// TwinCAT 3 PLC project Untitled1
// ProgramVersion: 3.1.4024.0
// libraries:
//   Tc2_Standard, * (Beckhoff Automation GmbH)
//   Tc2_System, * (Beckhoff Automation GmbH)
//   Tc3_Module, * (Beckhoff Automation GmbH)
//   VisuSymbols,3.5.10.0,System
// project tree:
//   DUTs/ T_State.TcDUT
//   / GlobalTextList.TcGTLO (not stored), PlcTask.TcTTO (not stored), task1.TcTTO (not stored), task2.TcTTO (not stored), task3.TcTTO (not stored), Task_4.TcTTO, Visualization Manager.TcVMO (not stored), Visualization.TcVIS (not stored)
//   GVLs/ GVL.TcGVL
//   POUs/ Main.TcPOU (not stored), PRG_BeerSession.TcPOU, PRG_GameSession.TcPOU, PRG_TrainTrip.TcPOU
// real-time tasks:
//   TASK PlcTask: cycle T#10ms, priority 20, ADS port 350
//   TASK Task 4: cycle T#10ms, priority 1, ADS port 351
//   TASK task1: cycle T#10ms, priority 21, ADS port 352
//   TASK task2: cycle T#10ms, priority 22, ADS port 353
//   TASK task3: cycle T#10ms, priority 23, ADS port 354

CONFIGURATION Untitled1
    RESOURCE PLC ON TwinCAT3
        TASK Task_4(INTERVAL := T#10ms, PRIORITY := 1);
        PROGRAM Main WITH Task_4 : Main;
        PROGRAM Main WITH Task_4 : Main;
    END_RESOURCE
END_CONFIGURATION

// ---- DUTs/T_State.TcDUT
TYPE T_State :
(
    WACHTEN,
    DRINKEN,
    LEEG,
    KLAAR
);
END_TYPE

// ---- GVLs/GVL.TcGVL
VAR_GLOBAL
    (* Treinreis *)
    ReisGestart      : BOOL := FALSE;
    OverstapBereikt  : BOOL := FALSE;
    Aangekomen       : BOOL := FALSE;

    (* Bier *)
    Biertjes         : UINT := 100;
	stefan_bier : UINT:= 0;
	wiebe_bier : UINT:= 0; 

    (* Spel *)
    SpelGestart      : BOOL := FALSE;
    Ronde            : UINT := 0;
	spelstop 		: BOOL:= FALSE; 

    (* Avond *)
    AvondKlaar       : BOOL := FALSE;
	IN: INT;
	koelkast_leeg : BOOL;  
	koelkast_vol : bool; 
	
END_VAR

// ---- POUs/PRG_BeerSession.TcPOU
PROGRAM PRG_BeerSession
VAR
    T_Biertje_stefan : TON;
	T_biertje_wiebe: ton; 
	T_biertje: ton; 
	koelkast : BOOL;
 State : T_State := WACHTEN;
END_VAR


CASE State OF

    // -------------------------
    WACHTEN:
    // -------------------------
        IF Aangekomen AND NOT AvondKlaar THEN
            IF biertjes > 0 THEN
                koelkast_vol := TRUE;
                koelkast_leeg := FALSE;
                State := DRINKEN;
            END_IF
        END_IF


    // -------------------------
    DRINKEN:
    // -------------------------
        // Timers alleen actief in deze state
        T_biertje_stefan(IN := TRUE, PT := T#3S);
        T_biertje_wiebe (IN := TRUE, PT := T#5S);

        // Stefan drinkt
        IF T_biertje_stefan.Q AND (biertjes > 0) THEN
            stefan_bier := stefan_bier + 1;
            biertjes := biertjes - 1;
            T_biertje_stefan(IN := FALSE);
        END_IF

        // Wibe drinkt
        IF T_biertje_wiebe.Q AND (biertjes > 0) THEN
            wiebe_bier := wiebe_bier + 1;
            biertjes := biertjes - 1;
            T_biertje_wiebe(IN := FALSE);
        END_IF

        // Overgang naar LEEG
        IF biertjes = 0 THEN
            State := LEEG;
        END_IF

        // Overgang naar KLAAR
        IF AvondKlaar THEN
            State := KLAAR;
        END_IF


    // -------------------------
    LEEG:
    // -------------------------
        koelkast_vol := FALSE;
        koelkast_leeg := TRUE;

        // Timers uit
        T_biertje_stefan(IN := FALSE);
        T_biertje_wiebe (IN := FALSE);

        IF AvondKlaar THEN
            State := KLAAR;
        END_IF


    // -------------------------
    KLAAR:
    // -------------------------
        koelkast_vol := FALSE;
        koelkast_leeg := TRUE;

        T_biertje_stefan(IN := FALSE);
        T_biertje_wiebe (IN := FALSE);

END_CASE

END_PROGRAM

// ---- POUs/PRG_GameSession.TcPOU
PROGRAM PRG_GameSession
VAR
    T_Ronde : TON;
END_VAR

IF  NOT SpelGestart AND koelkast_vol AND aangekomen THEN
    SpelGestart := TRUE;
	spelstop := FALSE; 
END_IF

IF SpelGestart = TRUE AND spelstop= FALSE AND (ronde<10) THEN 
    T_Ronde(IN := TRUE, PT := T#4S);

    IF T_Ronde.Q THEN
        Ronde := Ronde + 1;
        T_Ronde(IN := FALSE);
    END_IF
	IF koelkast_leeg= TRUE THEN
	spelstop:= TRUE; 
END_IF
	
	
END_IF

IF Ronde >= 10 THEN
    AvondKlaar := TRUE;
END_IF

END_PROGRAM

// ---- POUs/PRG_TrainTrip.TcPOU
PROGRAM PRG_TrainTrip
VAR
    T_Overstap : TON;
    T_Aankomst : TON;
END_VAR

IF NOT ReisGestart THEN
    ReisGestart := TRUE;
END_IF

(* Trein naar overstap *)
IF ReisGestart AND NOT OverstapBereikt THEN
    T_Overstap(IN := TRUE, PT := T#5S);

    IF T_Overstap.Q THEN
        OverstapBereikt := TRUE;
        T_Overstap(IN := FALSE);
    END_IF
END_IF

(* Trein naar eindbestemming *)
IF OverstapBereikt AND NOT Aangekomen THEN
    T_Aankomst(IN := TRUE, PT := T#5S);

    IF T_Aankomst.Q THEN
        Aangekomen := TRUE;
		koelkast_vol:=true; 
        T_Aankomst(IN := FALSE);
    END_IF
END_IF

END_PROGRAM
